FUNCTION_BLOCK CM_TUBELED_RGB IMPLEMENTS I_LED_RGB
VAR_OUTPUT
	Q_bColorRed AT %Q* : BOOL;
	Q_bColorGreen AT %Q* : BOOL;
	Q_bColorBlue AT %Q* : BOOL;
	Q_bColorWhite AT %Q* : BOOL;
END_VAR
VAR
	s_bColorRed : BOOL;
	s_bColorGreen : BOOL;
	s_bColorBlue : BOOL;
	s_bColorWhite : BOOL;	

	s_bFlash : BOOL;
	s_fbFlash : FB_Flash; 
END_VAR


s_fbFlash(
	i_bExcecute := TRUE,
	t_tOnTime := T#750MS,
	t_tOffTime := T#750MS,
	o_bQ => );

IF s_bFlash THEN
	Q_bColorRed := s_bColorRed AND s_fbFlash.o_bQ;
	Q_bColorGreen := s_bColorGreen AND s_fbFlash.o_bQ;
	Q_bColorBlue := s_bColorBlue AND s_fbFlash.o_bQ;
	Q_bColorWhite := s_bColorWhite AND s_fbFlash.o_bQ;
ELSE
	Q_bColorRed := s_bColorRed;
	Q_bColorGreen := s_bColorGreen;
	Q_bColorBlue := s_bColorBlue;
	Q_bColorWhite := s_bColorWhite;
END_IF

METHOD PUBLIC m_Blue : BOOL
VAR_INPUT
	i_bFlash : BOOL;
END_VAR

s_bColorRed := FALSE;
s_bColorGreen := FALSE;
s_bColorBlue := TRUE;
s_bColorWhite := FALSE;

s_bFlash := i_bFlash;
END_METHOD

METHOD PUBLIC m_Cyan : BOOL
VAR_INPUT
	i_bFlash : BOOL;
END_VAR

s_bColorRed := FALSE;
s_bColorGreen := TRUE;
s_bColorBlue := TRUE;
s_bColorWhite := FALSE;

s_bFlash := i_bFlash;
END_METHOD

METHOD PUBLIC m_Green : BOOL
VAR_INPUT
	i_bFlash : BOOL;
END_VAR

s_bColorRed := FALSE;
s_bColorGreen := TRUE;
s_bColorBlue := FALSE;
s_bColorWhite := FALSE;

s_bFlash := i_bFlash;
END_METHOD

METHOD PUBLIC m_Magenta : BOOL
VAR_INPUT
	i_bFlash : BOOL;
END_VAR

s_bColorRed := TRUE;
s_bColorGreen := FALSE;
s_bColorBlue := TRUE;
s_bColorWhite := FALSE;

s_bFlash := i_bFlash;
END_METHOD

METHOD PUBLIC m_Off : BOOL
VAR_INPUT
	i_bFlash : BOOL;
END_VAR

s_bColorRed := FALSE;
s_bColorGreen := FALSE;
s_bColorBlue := FALSE;
s_bColorWhite := FALSE;

s_bFlash := i_bFlash;
END_METHOD

METHOD PUBLIC m_Red : BOOL
VAR_INPUT
	i_bFlash : BOOL;
END_VAR

s_bColorRed := TRUE;
s_bColorGreen := FALSE;
s_bColorBlue := FALSE;
s_bColorWhite := FALSE;

s_bFlash := i_bFlash;
END_METHOD

METHOD PUBLIC m_White : BOOL
VAR_INPUT
	i_bFlash : BOOL;
END_VAR

s_bColorRed := FALSE;
s_bColorGreen := FALSE;
s_bColorBlue := FALSE;
s_bColorWhite := TRUE;

s_bFlash := i_bFlash;
END_METHOD

METHOD PUBLIC m_Yellow : BOOL
VAR_INPUT
	i_bFlash : BOOL;
END_VAR

s_bColorRed := TRUE;
s_bColorGreen := TRUE;
s_bColorBlue := FALSE;
s_bColorWhite := FALSE;

s_bFlash := i_bFlash;
END_METHOD

END_FUNCTION_BLOCK

(* stored: Version 1.1.0.1, ProductVersion 3.1.4024.12
   POU CM_TUBELED_RGB: Id {595df5ed-8c43-4c64-84d2-9ba9d4b953e6}, SpecialFunc None
   Method m_Blue: Id {811cd9fc-1a9c-4a3c-8f72-d33a4a0f6dcb}
   Method m_Cyan: Id {b5b902f2-be03-4a64-b2bb-64fe70cfdaef}
   Method m_Green: Id {ce16dd08-2cb3-42e7-b1f0-7228760bacfc}
   Method m_Magenta: Id {d186cc63-c07a-4047-a047-2a07b860d415}
   Method m_Off: Id {cbede21d-7f97-47a3-9390-3ee13ec52ca1}
   Method m_Red: Id {d35a4945-5d60-4fb4-9589-c3ea10729b99}
   Method m_White: Id {54898620-fb17-4318-ace3-ab1962baf179}
   Method m_Yellow: Id {d01841ca-9da5-44f7-a42f-be7c77a4e5f2} *)
